SUBAPPLICATION Checkbox_IDA_TO_AX_INIT_Force1 (* Checkbox_IDA_TO_AX_INIT (boot-stabiler AX-Pegel, startet TRUE bis zur ersten echten VT-Aenderung) + Q_NumericValue (F.22, erzwingt denselben NumberVariable-Wert bei FORTE-Start einmalig auf 1) zusammengefasst - Franz: 'gehoert ja zusammen', da beide dieselbe u16ObjId ansteuern/lesen. u16ObjId als Parameter fuer Wiederverwendung. *)
  (* Standard: 61499-2; Description: Copyright (c) 2026 Meisterschulen am Ostbahnhof This program and the accompanying materials are made available under the terms of the Eclipse Public License 2.0 which is available at https://www.eclipse.org/legal/epl-2.0/ SPDX-License-Identifier: EPL-2.0 *)
  (* Version 1.0, 2026-10-01, Franz Höpfinger, Meisterschulen am Ostbahnhof, initial implementation - aus Aufnahme_Automatik.SUB herausgeloest (Permit_Automatik + Q_NumericValue_Force1_Geschwindigkeitsregelung), u16ObjId als Parameter statt fest verdrahtet. *)
  PACKAGE MyLib_AX::sys;
  IMPORT isobus::UT::Q::const::IDs::ID_NULL;
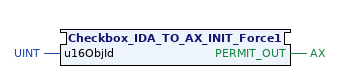
  VAR_INPUT
    u16ObjId : UINT := ID_NULL; (* Object ID der VT-Checkbox-NumberVariable (gleiches Objekt fuer Lesen und Force1-Schreiben) *)
  END_VAR
  PLUGS
    PERMIT_OUT : adapter::types::unidirectional::AX; (* Boot-stabiler Checkbox-Zustand (startet TRUE, folgt danach der echten VT-Checkbox) *)
  END_PLUGS
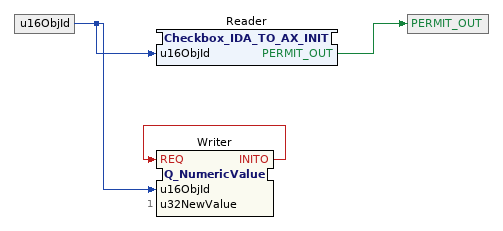
  FBS
    Writer : isobus::UT::Q::Q_NumericValue(u32NewValue := 1); (* Franz: 'soll bei INIT 1 werden' - fester FB-seitiger Einmalschreiber, NICHT die VT-Pool-InitialValue-Property. *)
  END_FBS
  SUBAPPS
    Reader : MyLib_AX::sys::Checkbox_IDA_TO_AX_INIT;
  END_SUBAPPS
  EVENT_CONNECTIONS
    Writer.INITO TO Writer.REQ;
  END_CONNECTIONS
  DATA_CONNECTIONS
    u16ObjId TO Reader.u16ObjId;
    u16ObjId TO Writer.u16ObjId;
  END_CONNECTIONS
  ADAPTER_CONNECTIONS
    Reader.PERMIT_OUT TO PERMIT_OUT;
  END_CONNECTIONS
END_SUBAPPLICATION
